FUNCTION_BLOCK "FB_ExecuteQuery2"
{ S7_Optimized_Access := 'TRUE' }
VERSION : 0.1
   VAR_INPUT
      query : String;
      params : Array[0..5] of Int;
      exec : Bool;
   END_VAR

   VAR
      Dispatch : Array[0..3] of Int;
      dataReady : Bool;
      dataError : Bool;
      noData : Bool;
      readyForNextQuery : Bool;
      queryCounter : Int;
      timeoutConnection {InstructionName := 'TON_TIME'; LibVersion := '1.0'; S7_SetPoint := 'False'} : TON_TIME;
      timeoutRetrayConnection {InstructionName := 'TON_TIME'; LibVersion := '1.0'} : TON_TIME;
      timeoutAbbandono {InstructionName := 'TON_TIME'; LibVersion := '1.0'} : TON_TIME;
   END_VAR

   VAR_TEMP
      queryTemp : String;
      i : Int;
   END_VAR


BEGIN
	//EXECUTE A QUERY AND WAIT THE RESULT!

	//check connection status
	//#timeoutConnection(IN := "InstLSql_Microsoft".status < 0 OR "InstLSql_Microsoft".status = 28672, //8602 / 7000
	//                   PT := t#1s);
	//"SqlConfig2".enableLSql := #timeoutConnection.Q ;


	//Check if is a SPECIAL QUERY

	REGION Sorveglianza connessione
	    // Nel canale 1 questa logica sta in FC_DBdata, che chiama i timer
	    // dell'istanza di FB6 dall'esterno. Qui non e' possibile: i timer di
	    // questo blocco, generato da sorgente esterno, sono tipi TON_TIME e
	    // non istanze di istruzione, e da un FC non si chiamano. Dentro il
	    // proprio FB la chiamata compila, quindi la sorveglianza vive qui.
	    // Differenza col canale 1: gira in coda allo scan (OB1 rete 7) invece
	    // che in testa (rete 1). Un ciclo di ritardo sul riarmo, irrilevante.
	    #timeoutConnection(IN := "SqlConfig2".enableLSql
	                       AND "SqlConfig2".diagnostics.status > 32770,
	                       PT := T#2s);
	    IF #timeoutConnection.Q THEN
	        "SqlConfig2".enableLSql := FALSE;
	    END_IF;

	    #timeoutRetrayConnection(IN := NOT "SqlConfig2".enableLSql,
	                             PT := T#1s);
	    IF #timeoutRetrayConnection.Q THEN
	        "SqlConfig2".enableLSql := TRUE;
	    END_IF;
	END_REGION

	IF #query = 'coordinate4ExtractTray' THEN
	    #queryTemp := CONCAT(IN1 := 'SELECT TRAY,X,Y,Z,X_ROT,Y_ROT,Z_ROT,APPROACH_TYPE,APPROACH_X,APPROACH_Y,APPROACH_Z from COORDINATES_FOR_EXTRACT where tray in (SELECT top(1) tray from COORDINATES_PIECES_TRAYS_4Robot where Order_ID=',
	                         IN2 := "INT_TO_STRING_WITHOUT_SIGN"(#params[0]),
	                         IN3 := ' AND status=',
	                         IN4 := "INT_TO_STRING_WITHOUT_SIGN"(#params[1]),
	                         IN5 := ' group BY tray)');
	    //--order BY tray desc
	ELSIF #query = 'coordinate4ExtractTrayWithID' THEN
	    #queryTemp := CONCAT(IN1 := 'SELECT TRAY,X,Y,Z,X_ROT,Y_ROT,Z_ROT from COORDINATES_FOR_EXTRACT where tray=',
	                         IN2 := "INT_TO_STRING_WITHOUT_SIGN"(#params[0]));
	ELSIF #query = 'tcpData' THEN
	    IF ("DB_Robot".Gripper_ID[1] <> 0 AND "DB_Robot".Gripper_ID[2] <> 0) THEN
	        #queryTemp := CONCAT(IN1 := 'select X_BODY+X_CLAW as X,Y_BODY+Y_CLAW as Y,Z_BODY+Z_CLAW as Z, VALVES, X_ROT, Y_ROT, Z_ROT from grippers where id in (',
	                             IN2 := "INT_TO_STRING_WITHOUT_SIGN"("DB_Robot".Gripper_ID[1]),
	                             IN3 := ',',
	                             IN4 := "INT_TO_STRING_WITHOUT_SIGN"("DB_Robot".Gripper_ID[2]),
	                             IN5 := ')');
	    ELSE
	        #queryTemp := CONCAT(IN1 := 'select X_BODY+X_CLAW as X,Y_BODY+Y_CLAW as Y,Z_BODY+Z_CLAW as Z, VALVES, X_ROT, Y_ROT, Z_ROT from grippers where id=',
	                             IN2 := "INT_TO_STRING_WITHOUT_SIGN"("DB_Robot".Gripper_ID[1]));
	    END_IF;
	ELSIF #query = 'coordinateMC' THEN
	    ;
	    (*SELECT SUB_POS ,X_PICK ,Y_PICK ,Z_PICK ,X_PLACE, Y_PLACE ,Z_PLACE ,X_ROT,Y_ROT,Z_ROT,APPROACh_type,APPROACH_X,APPROACH_Y,APPROACH_Z
	    from SmallBOX.dbo.COORDINATES_PIECES_MC
	    where MC =2
	    *)
	ELSIF #query = 'updateTrayExtract' THEN
	    #queryTemp := CONCAT(IN1 := 'UPDATE TRAY SET [EXTRACT]=',
	                         IN2 := "INT_TO_STRING_WITHOUT_SIGN"(#params[0]),
	                         IN3 := ' WHERE FLOOR_MAG=',
	                         IN4 := "INT_TO_STRING_WITHOUT_SIGN"(#params[1]));
	ELSE
	    #queryTemp := #query;
	END_IF;


	CASE #Dispatch["_master"] OF
	    0:  //nothing to do
	        // GUARDIA DI RIPRISTINO (5/9): a riposo il buffer DEVE essere vuoto.
	        // Se qualcuno azzera Dispatch dall'esterno (resetDispatcher di FB7,
	        // forzature da watch) senza svuotare sqlCommands[0], il ponte resta
	        // occupato per sempre: nessun richiedente riesce piu' a scrivere la
	        // propria query perche' tutti controllano sqlCommands[0] = ''.
	        // Sintomo visto il 5/9: Dispatch a 0, readyForNextQuery TRUE,
	        // dataReady FALSE e buffer pieno — cella ferma senza errori.
	        IF "SqlCommands2".sqlCommands[0] <> '' THEN
	            "SqlCommands2".sqlCommands[0] := '';
	        END_IF;

	        IF #exec THEN
	            #Dispatch["_master"] := 10;
	            #readyForNextQuery := FALSE;
	            #dataError := false;
	            #noData := false;
	            #dataReady := false;
	            "SqlData2".data.rowCount := 0;
	        END_IF;

	    10: // write query
	        IF (LEN(#queryTemp) > 1 AND "SqlConfig2".diagnostics.status >= 0 AND "SqlConfig2".enableLSql) THEN
	            "SqlCommands2".sqlCommands[0] := #queryTemp;
	            "SqlCommands2".currentSqlCommand := 0;

	            #Dispatch["_master"] := 20;
	        END_IF;

	    20: // execute query
	        "SqlConfig2".executeSqlCommand := TRUE;
	        #Dispatch["_master"] := 30;

	    30: // wait result
	        IF "SqlTdsReceive2".tdsTelegramArrayLength > 0
	            AND NOT "SqlConfig2".executeSqlCommand THEN
	            #queryCounter := #queryCounter + 1;

	            #Dispatch["_master"] := 35;
	        END_IF;

	    35: //wait syncro from cycle plc
	        // TIMEOUT DI ABBANDONO (5/9): se il richiedente muore prima di leggere
	        // il risultato (errore, reset, catena che cambia stato) nessuno alza
	        // readyForNextQuery e il ponte resta appeso qui bloccando tutta la
	        // cella. Dopo 60s si libera da solo: il risultato va perso, ma il
	        // ponte torna disponibile invece di piantare l'impianto.
	        #timeoutAbbandono(IN := TRUE,
	                          PT := T#60s);

	        IF #readyForNextQuery OR #timeoutAbbandono.Q THEN
	            #timeoutAbbandono(IN := FALSE,
	                              PT := T#60s);

	            //save last query into log
	            FOR #i := 5 TO 1 BY -1 DO
	                "SqlCommands2".sqlCommands[#i] := "SqlCommands2".sqlCommands[#i - 1];
	            END_FOR;
	            "SqlCommands2".sqlCommands[0] := '';

	            #readyForNextQuery := TRUE;
	            #Dispatch["_master"] := 0;
	        END_IF;
	    ELSE
	        // stato non previsto (forzatura, corruzione): torno a riposo pulito
	        "SqlCommands2".sqlCommands[0] := '';
	        #readyForNextQuery := TRUE;
	        #Dispatch["_master"] := 0;
	END_CASE;


	// dataReady: SOLO allo stato 35 il risultato e' effettivamente disponibile.
	#dataReady := #Dispatch["_master"] = 35;

	#noData := "SqlData2".data.rowCount = 0;

	// dataError: SOLO errore vero del ponte.
	// RIMOSSO il termine LEN(#queryTemp) = 0: #queryTemp e' la temporanea
	// ricalcolata a OGNI chiamata dal parametro query, e OB1 Network 7 passa
	// stringa vuota quando nessuno ha richieste pendenti. Cosi' dataError
	// diventava vero su un risultato perfettamente valido, appena il flag del
	// richiedente cadeva (visto 4/9: errore al parsing con SqlData corretto).
	#dataError := "SqlConfig2".diagnostics.status > 8000;
END_FUNCTION_BLOCK

